FUNCTION_BLOCK Door
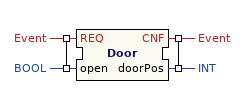
  EVENT_INPUT
    REQ WITH open;
  END_EVENT
  EVENT_OUTPUT
    CNF WITH doorPos;
  END_EVENT
  VAR_INPUT
    open : BOOL;
  END_VAR
  VAR_OUTPUT
    doorPos : INT;
  END_VAR
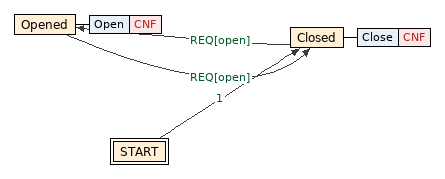
  EC_STATES
    START;
    Opened : Open -> CNF;
    Closed : Close -> CNF;
  END_STATES
  EC_TRANSITIONS
    START TO Closed := 1;
    Closed TO Opened := REQ[open];
    Opened TO Closed := REQ[open];
  END_TRANSITIONS
  ALGORITHM Open IN ST:
doorPos := 10;&#38;#10;
  END_ALGORITHM
  ALGORITHM Close IN ST:
doorPos := 0;&#38;#10;
  END_ALGORITHM
END_FUNCTION_BLOCK
